Fanuc KAREL source: ka00012.KL

PROGRAM KA00012
%STACKSIZE=65535
%PRIORITY=65535
%NOLOCKGROUP
VAR
SRC : INTEGER
-- UNRESOLVED DECLARATIONS (source type spelling not recovered)
-- DST : ARRAY[2] OF TYPE_0x0017 (type_u16=0x2017)
BEGIN
SRC=2
-- UNRESOLVED_PC line 8 opcodes [21 22 9D 33 B4] marker_code=16
END KA00012
